% RSLogix 500 project simular_HMI.RSS, saved by version 8.30.00.15 %
PROJECT "S3011222"    % processor: Bul.1763 MicroLogix 1100 Series B %

PROGRAM FILES
  LAD 2   14 rungs

DATA FILES
  O0 OUTPUT  6 elements
  I1 INPUT  12 elements
  S2 STATUS  66 elements
  B3 BINARY  1 elements
  T4 TIMER  1 elements
  C5 COUNTER  1 elements
  R6 CONTROL  1 elements
  N7 INTEGER  10 elements
  F8 FLOAT  9 elements
  PD9   1 elements

LADDER 2
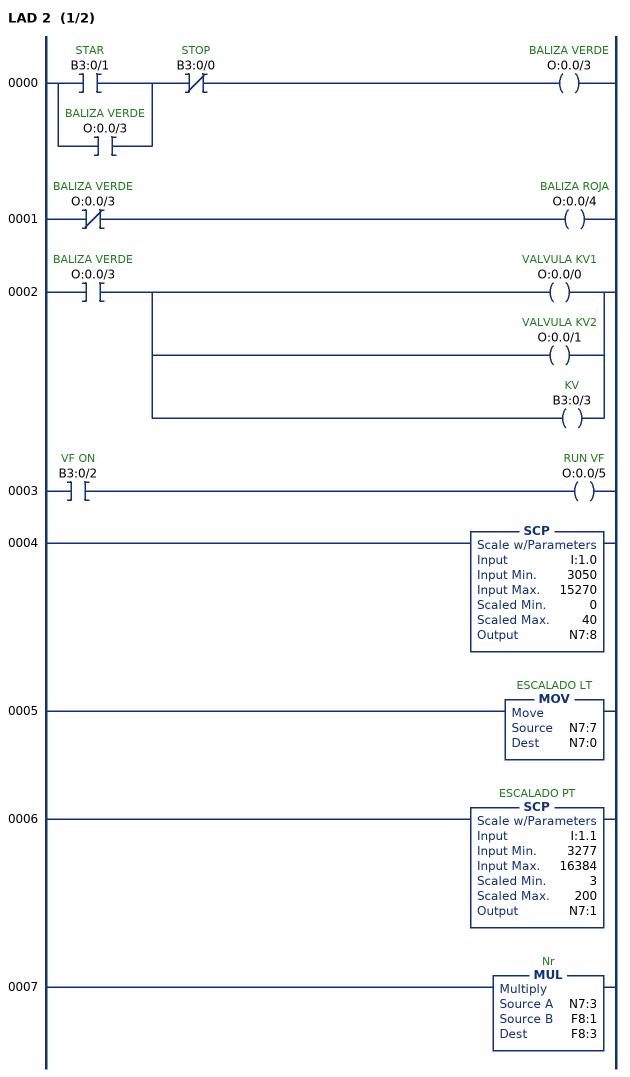
% Rung: 0 %
SOR BST XIC B3:0/1 NXB XIC O:0.0/3 BND XIO B3:0/0 OTE O:0.0/3 EOR
%   B3:0/1  "STAR" %
%   O:0.0/3  "BALIZA VERDE" %
%   B3:0/0  "STOP" %
% Rung: 1 %
SOR XIO O:0.0/3 OTE O:0.0/4 EOR
%   O:0.0/3  "BALIZA VERDE" %
%   O:0.0/4  "BALIZA ROJA" %
% Rung: 2 %
SOR XIC O:0.0/3 BST OTE O:0.0/0 NXB BST OTE O:0.0/1 NXB OTE B3:0/3 BND BND EOR
%   O:0.0/3  "BALIZA VERDE" %
%   O:0.0/0  "VALVULA KV1" %
%   O:0.0/1  "VALVULA KV2" %
%   B3:0/3  "KV" %
% Rung: 3 %
SOR XIC B3:0/2 OTE O:0.0/5 EOR
%   B3:0/2  "VF ON" %
%   O:0.0/5  "RUN VF" %
% Rung: 4 %
SOR SCP I:1.0 3050 15270 0 40 N7:8 EOR
%   I:1.0  "LT" %
% Rung: 5 %
SOR MOV N7:7 N7:0 EOR
%   N7:0  "ESCALADO LT" %
% Rung: 6 %
SOR SCP I:1.1 3277 16384 3 200 N7:1 EOR
%   I:1.1  "PT" %
%   N7:1  "ESCALADO PT" %
% Rung: 7 %
SOR MUL N7:3 F8:1 F8:3 EOR
%   N7:3  "SET POINT" %
%   F8:1  "N" %
%   F8:3  "Nr" %

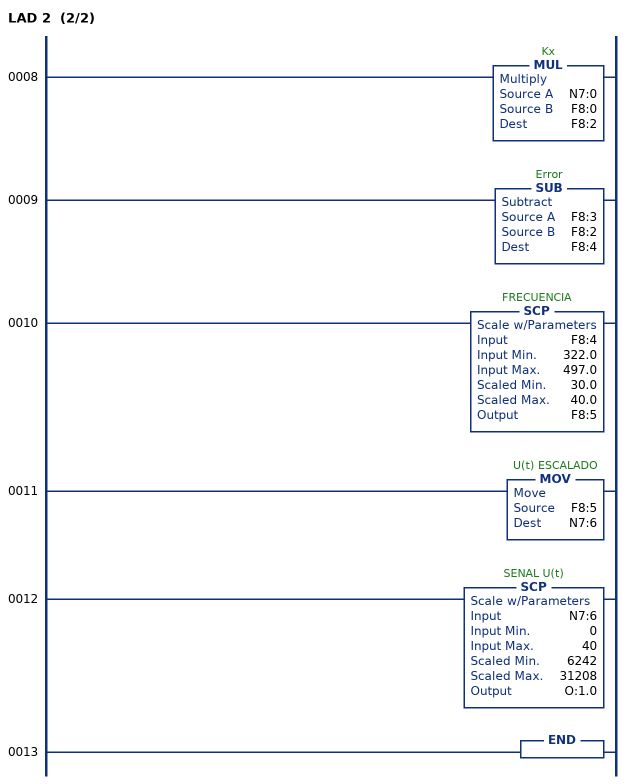
% Rung: 8 %
SOR MUL N7:0 F8:0 F8:2 EOR
%   N7:0  "ESCALADO LT" %
%   F8:0  "K" %
%   F8:2  "Kx" %
% Rung: 9 %
SOR SUB F8:3 F8:2 F8:4 EOR
%   F8:3  "Nr" %
%   F8:2  "Kx" %
%   F8:4  "Error" %
% Rung: 10 %
SOR SCP F8:4 322.0 497.0 30.0 40.0 F8:5 EOR
%   F8:4  "Error" %
%   F8:5  "FRECUENCIA" %
% Rung: 11 %
SOR MOV F8:5 N7:6 EOR
%   F8:5  "FRECUENCIA" %
%   N7:6  "U(t) ESCALADO" %
% Rung: 12 %
SOR SCP N7:6 0 40 6242 31208 O:1.0 EOR
%   N7:6  "U(t) ESCALADO" %
%   O:1.0  "SENAL U(t)" %
% Rung: 13 %
SOR END EOR

OTHER DOCUMENTED ADDRESSES
  I:0.0/3  "ENCENDIDO"
  I:0.0/4  "APAGADO"
  I:0.0/5  "ENCENDER VARIADOR"
  N7:2  "ERROR"
  N7:4  "Nr(t)"
  N7:5  "Kx(t)"
  PD9:0.2  "REFERENCIA"
  PD9:0.3  "Kc"
  PD9:0.4  "Ti"
  PD9:0.5  "Td"

DATA TABLE (non-zero values as saved)
DATA N7
% N7:0 % 0 1 0 20 0 0 52 0 20 6
DATA F8
% F8:0 % 29.3165 35.5556 0 711.112 711.112
% F8:5 % 52.23497 0 0 0
